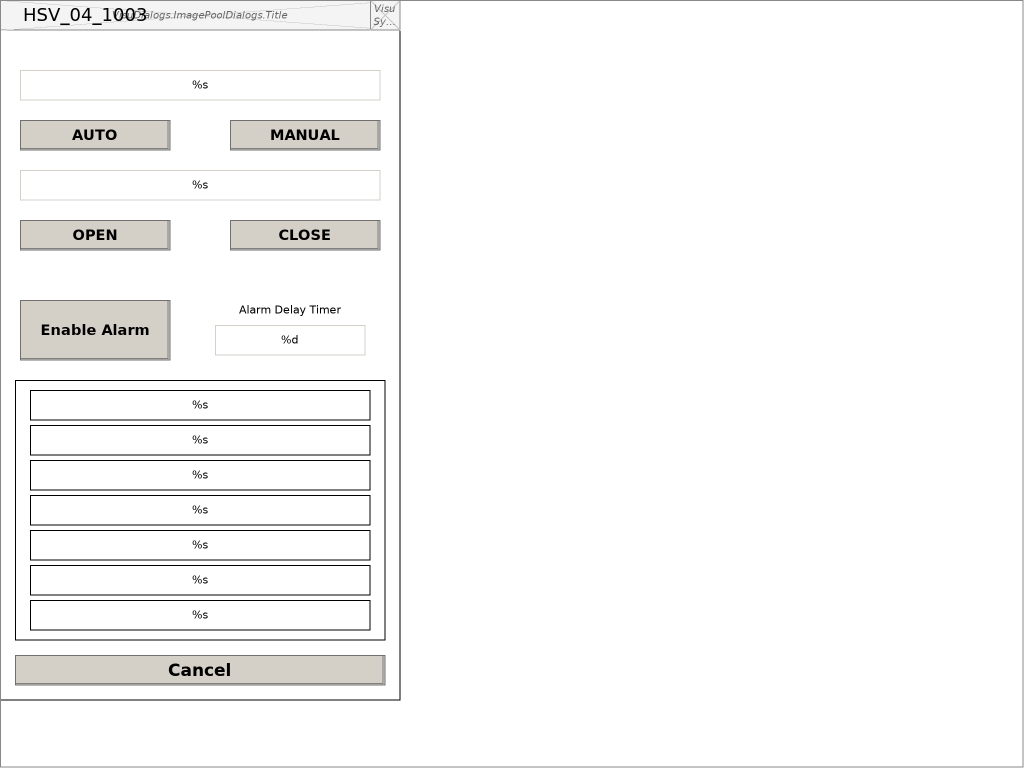
VISUALIZATION HSV_04_1003  // 1024x768
    Rectangle (0,0 400x700)
    Button (20,120 150x30), "AUTO"
        tap progHSVCntrl.HSV_04_1003.AutoReq
    Button (230,120 150x30), "MANUAL"
        tap progHSVCntrl.HSV_04_1003.ManReq
    Button (20,220 150x30), "OPEN"
        tap progHSVCntrl.HSV_04_1003.ManOpenReq
    Button (230,220 150x30), "CLOSE"
        tap progHSVCntrl.HSV_04_1003.ManCloseReq
    Textfield (20,70 360x30), "%s", text variable: progHSVCntrl.HSV_04_1003.strAutoMan
    Textfield (20,170 360x30), "%s", text variable: progHSVCntrl.HSV_04_1003.strOpenTravClose
    Button (20,300 150x60), "Enable Alarm"
        toggle progHSVCntrl.HSV_04_1003.EnableAlarm
    Textfield (215,325 150x30), "%d", text variable: progHSVCntrl.HSV_04_1003.AlarmDelayTime
    Label (215,295 150x30), "Alarm Delay Timer"
    Image (0,0 400x30), image: VisuDialogs.ImagePoolDialogs.Title
    Group (370,0 30x30)
        OnMouseClick: CloseDialog Dialog=HSV_04_1003, Result=OK, NumpadKeypadSet=True
        RoundedRectangle (0,0 30x30)
        Image (0,0 30x30), image: VisuSymbols.Symbols.Wrong
    Rectangle (15,380 370x260)
    RoundedRectangle (30,390 340x30), "%s", text variable: progHSVCntrl.HSV_04_1003.strInterlock_1
    RoundedRectangle (30,425 340x30), "%s", text variable: progHSVCntrl.HSV_04_1003.strInterlock_2
    RoundedRectangle (30,460 340x30), "%s", text variable: progHSVCntrl.HSV_04_1003.strInterlock_3
    RoundedRectangle (30,495 340x30), "%s", text variable: progHSVCntrl.HSV_04_1003.strInterlock_4
    RoundedRectangle (30,530 340x30), "%s", text variable: progHSVCntrl.HSV_04_1003.strInterlock_5
    RoundedRectangle (30,565 340x30), "%s", text variable: progHSVCntrl.HSV_04_1003.strInterlock_6
    RoundedRectangle (30,600 340x30), "%s", text variable: progHSVCntrl.HSV_04_1003.strInterlock_7
    Button (15,655 370x30), "Cancel"
        OnMouseClick: CloseDialog Dialog=HSV_04_1003, Result=OK, NumpadKeypadSet=True
    Label (20,0 210x30), "HSV_04_1003"
END_VISUALIZATION

// ---- VISUs/Diag/HSV/HSV_04_1004.TcVIS
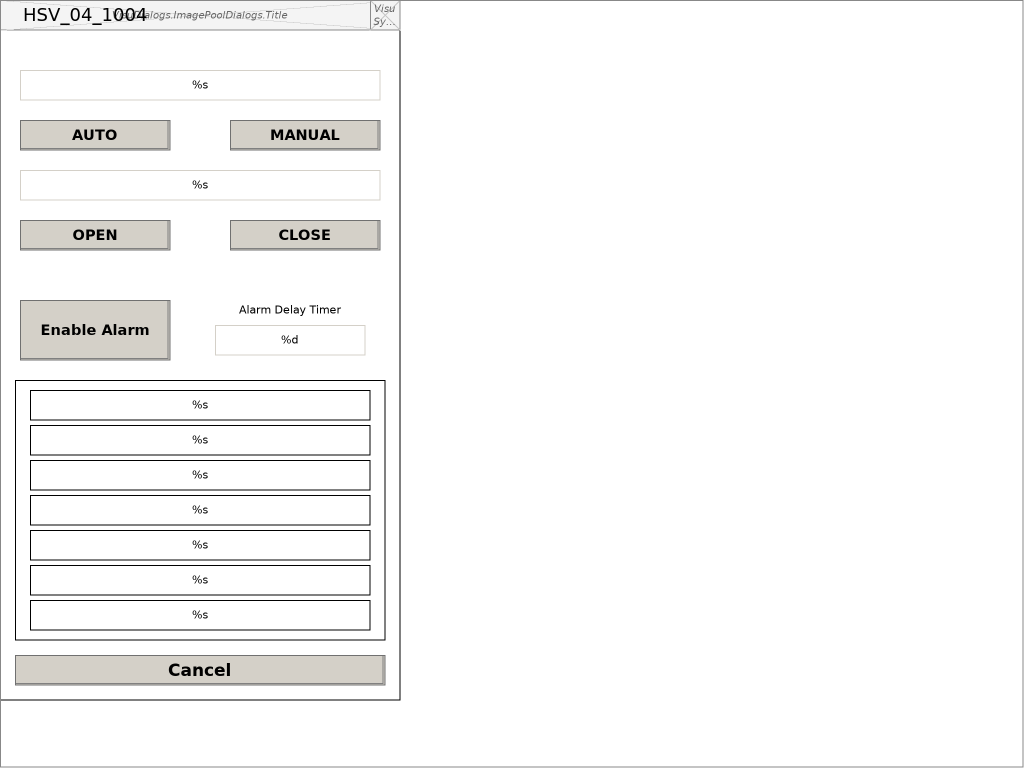
VISUALIZATION HSV_04_1004  // 1024x768
    Rectangle (0,0 400x700)
    Button (20,120 150x30), "AUTO"
        tap progHSVCntrl.HSV_04_1004.AutoReq
    Button (230,120 150x30), "MANUAL"
        tap progHSVCntrl.HSV_04_1004.ManReq
    Button (20,220 150x30), "OPEN"
        tap progHSVCntrl.HSV_04_1004.ManOpenReq
    Button (230,220 150x30), "CLOSE"
        tap progHSVCntrl.HSV_04_1004.ManCloseReq
    Textfield (20,70 360x30), "%s", text variable: progHSVCntrl.HSV_04_1004.strAutoMan
    Textfield (20,170 360x30), "%s", text variable: progHSVCntrl.HSV_04_1004.strOpenTravClose
    Button (20,300 150x60), "Enable Alarm"
        toggle progHSVCntrl.HSV_04_1004.EnableAlarm
    Textfield (215,325 150x30), "%d", text variable: progHSVCntrl.HSV_04_1004.AlarmDelayTime
    Label (215,295 150x30), "Alarm Delay Timer"
    Image (0,0 400x30), image: VisuDialogs.ImagePoolDialogs.Title
    Group (370,0 30x30)
        OnMouseClick: CloseDialog Dialog=HSV_04_1004, Result=OK, NumpadKeypadSet=True
        RoundedRectangle (0,0 30x30)
        Image (0,0 30x30), image: VisuSymbols.Symbols.Wrong
    Rectangle (15,380 370x260)
    RoundedRectangle (30,390 340x30), "%s", text variable: progHSVCntrl.HSV_04_1004.strInterlock_1
    RoundedRectangle (30,425 340x30), "%s", text variable: progHSVCntrl.HSV_04_1004.strInterlock_2
    RoundedRectangle (30,460 340x30), "%s", text variable: progHSVCntrl.HSV_04_1004.strInterlock_3
    RoundedRectangle (30,495 340x30), "%s", text variable: progHSVCntrl.HSV_04_1004.strInterlock_4
    RoundedRectangle (30,530 340x30), "%s", text variable: progHSVCntrl.HSV_04_1004.strInterlock_5
    RoundedRectangle (30,565 340x30), "%s", text variable: progHSVCntrl.HSV_04_1004.strInterlock_6
    RoundedRectangle (30,600 340x30), "%s", text variable: progHSVCntrl.HSV_04_1004.strInterlock_7
    Button (15,655 370x30), "Cancel"
        OnMouseClick: CloseDialog Dialog=HSV_04_1004, Result=OK, NumpadKeypadSet=True
    Label (20,0 210x30), "HSV_04_1004"
END_VISUALIZATION

// ---- VISUs/Diag/HSV/HSV_04_1005.TcVIS
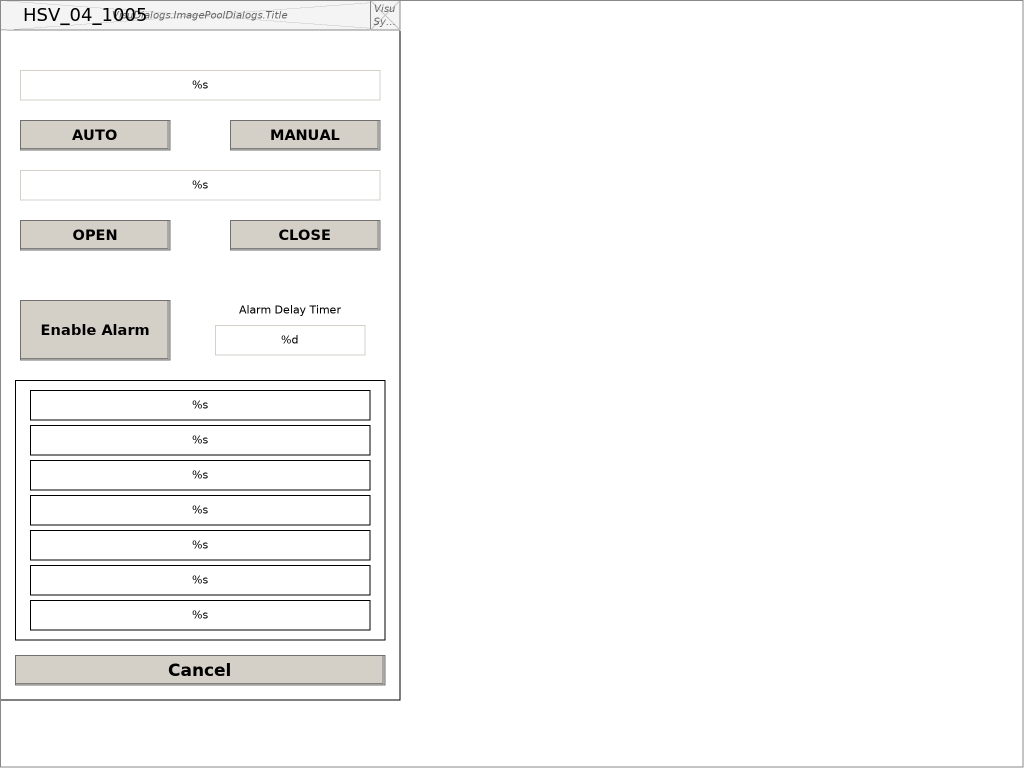
VISUALIZATION HSV_04_1005  // 1024x768
    Rectangle (0,0 400x700)
    Button (20,120 150x30), "AUTO"
        tap progHSVCntrl.HSV_04_1005.AutoReq
    Button (230,120 150x30), "MANUAL"
        tap progHSVCntrl.HSV_04_1005.ManReq
    Button (20,220 150x30), "OPEN"
        tap progHSVCntrl.HSV_04_1005.ManOpenReq
    Button (230,220 150x30), "CLOSE"
        tap progHSVCntrl.HSV_04_1005.ManCloseReq
    Textfield (20,70 360x30), "%s", text variable: progHSVCntrl.HSV_04_1005.strAutoMan
    Textfield (20,170 360x30), "%s", text variable: progHSVCntrl.HSV_04_1005.strOpenTravClose
    Button (20,300 150x60), "Enable Alarm"
        toggle progHSVCntrl.HSV_04_1005.EnableAlarm
    Textfield (215,325 150x30), "%d", text variable: progHSVCntrl.HSV_04_1005.AlarmDelayTime
    Label (215,295 150x30), "Alarm Delay Timer"
    Image (0,0 400x30), image: VisuDialogs.ImagePoolDialogs.Title
    Group (370,0 30x30)
        OnMouseClick: CloseDialog Dialog=HSV_04_1005, Result=OK, NumpadKeypadSet=True
        RoundedRectangle (0,0 30x30)
        Image (0,0 30x30), image: VisuSymbols.Symbols.Wrong
    Rectangle (15,380 370x260)
    RoundedRectangle (30,390 340x30), "%s", text variable: progHSVCntrl.HSV_04_1005.strInterlock_1
    RoundedRectangle (30,425 340x30), "%s", text variable: progHSVCntrl.HSV_04_1005.strInterlock_2
    RoundedRectangle (30,460 340x30), "%s", text variable: progHSVCntrl.HSV_04_1005.strInterlock_3
    RoundedRectangle (30,495 340x30), "%s", text variable: progHSVCntrl.HSV_04_1005.strInterlock_4
    RoundedRectangle (30,530 340x30), "%s", text variable: progHSVCntrl.HSV_04_1005.strInterlock_5
    RoundedRectangle (30,565 340x30), "%s", text variable: progHSVCntrl.HSV_04_1005.strInterlock_6
    RoundedRectangle (30,600 340x30), "%s", text variable: progHSVCntrl.HSV_04_1005.strInterlock_7
    Button (15,655 370x30), "Cancel"
        OnMouseClick: CloseDialog Dialog=HSV_04_1005, Result=OK, NumpadKeypadSet=True
    Label (20,0 210x30), "HSV_04_1005"
END_VISUALIZATION

// ---- VISUs/Diag/SCA/SCA_04_0100.TcVIS
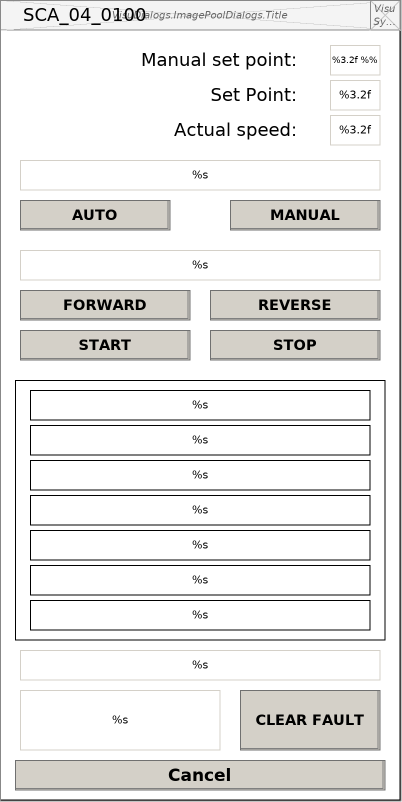
VISUALIZATION SCA_04_0100  // 402x802
    Rectangle (0,0 400x800)
    Button (20,200 150x30), "AUTO"
        tap progSCACntrl.SCA_04_0100.AutoReq
    Button (230,200 150x30), "MANUAL"
        tap progSCACntrl.SCA_04_0100.ManReq
    Button (20,290 170x30), "FORWARD"
        OnMouseClick: execute { progSCACntrl.SCA_04_0100.ManDirection := 0; }
    Button (210,290 170x30), "REVERSE"
        OnMouseClick: execute { progSCACntrl.SCA_04_0100.ManDirection := 1; }
    Textfield (20,160 360x30), "%s", text variable: progSCACntrl.SCA_04_0100.strAutoMan
    Textfield (20,250 360x30), "%s", text variable: progSCACntrl.SCA_04_0100.strStopTravRun
    Image (0,0 400x30), image: VisuDialogs.ImagePoolDialogs.Title
    Group (370,0 30x30)
        RoundedRectangle (0,0 30x30)
        Image (0,0 30x30), image: VisuSymbols.Symbols.Wrong
    Rectangle (15,380 370x260)
    RoundedRectangle (30,390 340x30), "%s", text variable: progSCACntrl.SCA_04_0100.strInterlock_1
    RoundedRectangle (30,425 340x30), "%s", text variable: progSCACntrl.SCA_04_0100.strInterlock_2
    RoundedRectangle (30,460 340x30), "%s", text variable: progSCACntrl.SCA_04_0100.strInterlock_3
    RoundedRectangle (30,495 340x30), "%s", text variable: progSCACntrl.SCA_04_0100.strInterlock_4
    RoundedRectangle (30,530 340x30), "%s", text variable: progSCACntrl.SCA_04_0100.strInterlock_5
    RoundedRectangle (30,565 340x30), "%s", text variable: progSCACntrl.SCA_04_0100.strInterlock_6
    RoundedRectangle (30,600 340x30), "%s", text variable: progSCACntrl.SCA_04_0100.strInterlock_7
    Button (15,760 370x30), "Cancel"
    Label (0,80 300x30), "Set Point:"
    Textfield (330,80 50x30), "%3.2f", text variable: progSCACntrl.SCA_04_0100.CommandSpeed
    Label (0,45 300x30), "Manual set point:"
    Textfield (330,45 50x30), "%3.2f %%", text variable: progSCACntrl.SCA_04_0100.ManSpeed
        OnMouseClick: write the text variable via VisuDialogs.Numpad, min progSCACntrl.SCA_04_0100.EngMin, max progSCACntrl.SCA_04_0100.EngMax, format %3.2f
    Label (0,115 300x30), "Actual speed:"
    Textfield (330,115 50x30), "%3.2f", text variable: progSCACntrl.SCA_04_0100.ActualSpeed
    Label (20,0 210x30), "SCA_04_0100"
    Button (20,330 170x30), "START"
        tap progSCACntrl.SCA_04_0100.ManStart
    Button (210,330 170x30), "STOP"
        tap progSCACntrl.SCA_04_0100.ManStop
    Textfield (20,650 360x30), "%s", text variable: progSCACntrl.SCA_04_0100.strAlmDesc
    Textfield (20,690 200x60), "%s", text variable: progSCACntrl.SCA_04_0100.strOKFault
    Button (240,690 140x60), "CLEAR FAULT"
        tap progSCACntrl.SCA_04_0100.ClearFlt
END_VISUALIZATION

// ---- VISUs/Screens/Overview.TcVIS
VISUALIZATION Overview  // 2x2
END_VISUALIZATION

// ---- VISUs/Screens/Vacuum_C1.TcVIS
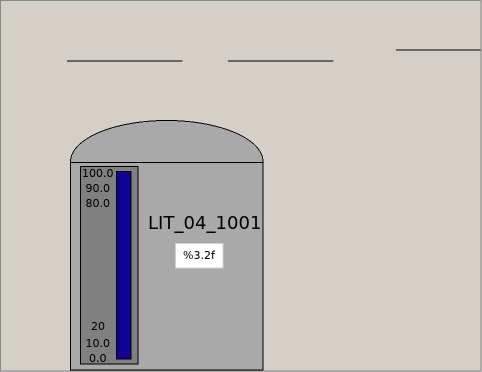
VISUALIZATION Vacuum_C1  // 482x372
    Line (182,61) (67,61)
    Line (333,61) (228,61)
    Line (480,50) (396,50)
    Group (70,120 200x250)
        Ellipse (0,0 193x83)
        Rectangle (0,42 193x208)
        Rectangle (10,46 58x198)
        Rectangle (46,51 15x188)
        Label (10,231 36x15), "0.0"
        Label (10,46 36x15), "100.0"
        Label (10,61 36x15), "90.0"
        Label (10,76 36x15), "80.0"
        Label (10,216 36x15), "10.0"
        Label (10,199 36x15), "20"
        Label (70,88 130x30), "LIT_04_1001"
        Textfield (105,123 48x25), "%3.2f", text variable: progLITCntrl.LIT_04_1001.Level
            OnMouseClick: write progLITCntrl.LIT_04_1001.Level via VisuDialogs.NumpadExtended, min 0.0, max 100.0
END_VISUALIZATION

// ---- VISUs/Templates/Diag/visuFCVDiag.TcVIS
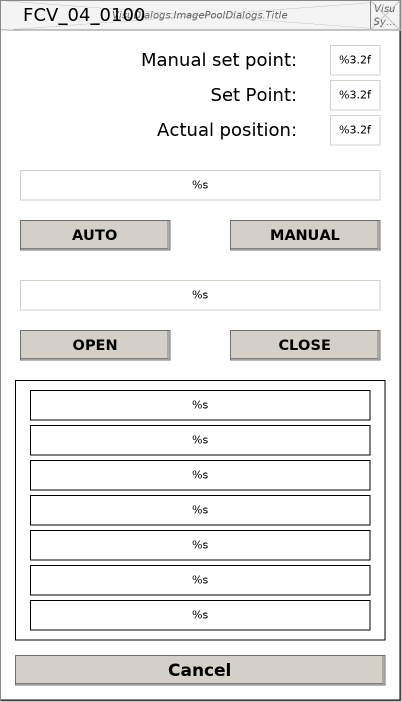
VISUALIZATION visuFCVDiag  // 402x702
    Rectangle (0,0 400x700)
    Button (20,220 150x30), "AUTO"
        tap progFCVCntrl.FCV_04_0100.AutoReq
    Button (230,220 150x30), "MANUAL"
        tap progFCVCntrl.FCV_04_0100.ManReq
    Button (20,330 150x30), "OPEN"
        tap progFCVCntrl.FCV_04_0100.ManOpenReq
    Button (230,330 150x30), "CLOSE"
        tap progFCVCntrl.FCV_04_0100.ManCloseReq
    Textfield (20,170 360x30), "%s", text variable: progFCVCntrl.FCV_04_0100.strAutoMan
    Textfield (20,280 360x30), "%s", text variable: progFCVCntrl.FCV_04_0100.strOpenTravClose
    Image (0,0 400x30), image: VisuDialogs.ImagePoolDialogs.Title
    Group (370,0 30x30)
        RoundedRectangle (0,0 30x30)
        Image (0,0 30x30), image: VisuSymbols.Symbols.Wrong
    Rectangle (15,380 370x260)
    RoundedRectangle (30,390 340x30), "%s", text variable: progFCVCntrl.FCV_04_0100.strInterlock_1
    RoundedRectangle (30,425 340x30), "%s", text variable: progFCVCntrl.FCV_04_0100.strInterlock_2
    RoundedRectangle (30,460 340x30), "%s", text variable: progFCVCntrl.FCV_04_0100.strInterlock_3
    RoundedRectangle (30,495 340x30), "%s", text variable: progFCVCntrl.FCV_04_0100.strInterlock_4
    RoundedRectangle (30,530 340x30), "%s", text variable: progFCVCntrl.FCV_04_0100.strInterlock_5
    RoundedRectangle (30,565 340x30), "%s", text variable: progFCVCntrl.FCV_04_0100.strInterlock_6
    RoundedRectangle (30,600 340x30), "%s", text variable: progFCVCntrl.FCV_04_0100.strInterlock_7
    Button (15,655 370x30), "Cancel"
    Label (0,80 300x30), "Set Point:"
    Textfield (330,80 50x30), "%3.2f", text variable: progFCVCntrl.FCV_04_0100.CmdSpOut
    Label (0,45 300x30), "Manual set point:"
    Textfield (330,45 50x30), "%3.2f", text variable: progFCVCntrl.FCV_04_0100.ManSP
        OnMouseClick: write progFCVCntrl.FCV_04_0100.ManSP via VisuDialogs.NumpadExtended
    Label (0,115 300x30), "Actual position:"
    Textfield (330,115 50x30), "%3.2f", text variable: progFCVCntrl.FCV_04_0100.ActPos
    Label (20,0 210x30), "FCV_04_0100"
END_VISUALIZATION

// ---- VISUs/Templates/Diag/visuHSVDiag.TcVIS
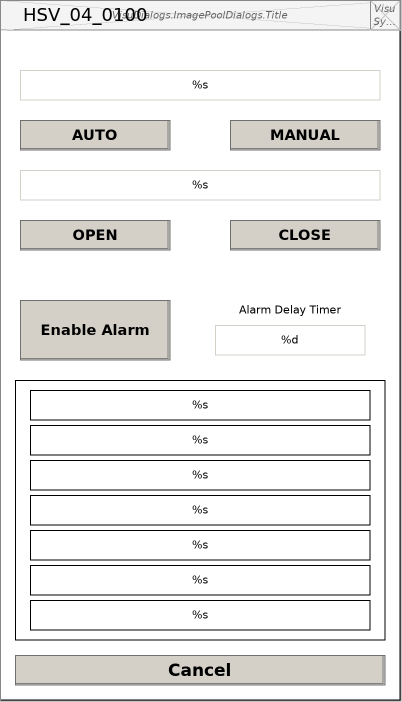
VISUALIZATION visuHSVDiag  // 402x702
    Rectangle (0,0 400x700)
    Button (20,120 150x30), "AUTO"
        tap progHSVCntrl.HSV_04_0100.AutoReq
    Button (230,120 150x30), "MANUAL"
        tap progHSVCntrl.HSV_04_0100.ManReq
    Button (20,220 150x30), "OPEN"
        tap progHSVCntrl.HSV_04_0100.ManOpenReq
    Button (230,220 150x30), "CLOSE"
        tap progHSVCntrl.HSV_04_0100.ManCloseReq
    Textfield (20,70 360x30), "%s", text variable: progHSVCntrl.HSV_04_0100.strAutoMan
    Textfield (20,170 360x30), "%s", text variable: progHSVCntrl.HSV_04_0100.strOpenTravClose
    Button (20,300 150x60), "Enable Alarm"
        toggle progHSVCntrl.HSV_04_0100.EnableAlarm
    Textfield (215,325 150x30), "%d"
    Label (215,295 150x30), "Alarm Delay Timer"
    Image (0,0 400x30), image: VisuDialogs.ImagePoolDialogs.Title
    Group (370,0 30x30)
        RoundedRectangle (0,0 30x30)
        Image (0,0 30x30), image: VisuSymbols.Symbols.Wrong
    Rectangle (15,380 370x260)
    RoundedRectangle (30,390 340x30), "%s", text variable: progHSVCntrl.HSV_04_0100.strInterlock_1
    RoundedRectangle (30,425 340x30), "%s", text variable: progHSVCntrl.HSV_04_0100.strInterlock_2
    RoundedRectangle (30,460 340x30), "%s", text variable: progHSVCntrl.HSV_04_0100.strInterlock_3
    RoundedRectangle (30,495 340x30), "%s", text variable: progHSVCntrl.HSV_04_0100.strInterlock_4
    RoundedRectangle (30,530 340x30), "%s", text variable: progHSVCntrl.HSV_04_0100.strInterlock_5
    RoundedRectangle (30,565 340x30), "%s", text variable: progHSVCntrl.HSV_04_0100.strInterlock_6
    RoundedRectangle (30,600 340x30), "%s", text variable: progHSVCntrl.HSV_04_0100.strInterlock_7
    Button (15,655 370x30), "Cancel"
    Label (20,0 210x30), "HSV_04_0100"
END_VISUALIZATION

// ---- VISUs/Templates/Diag/visuLITDiag.TcVIS
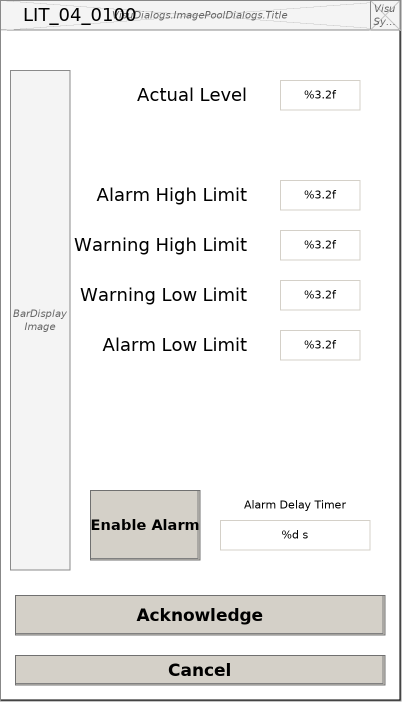
VISUALIZATION visuLITDiag  // 402x702
    Rectangle (0,0 400x700)
    Textfield (280,180 80x30), "%3.2f", text variable: progLITCntrl.LIT_04_0100.HHLimit
    Button (90,490 110x70), "Enable Alarm"
        toggle progHSVCntrl.HSV_04_0100.EnableAlarm
    Textfield (220,520 150x30), "%d s"
    Label (220,490 150x30), "Alarm Delay Timer"
    Image (0,0 400x30), image: VisuDialogs.ImagePoolDialogs.Title
    Group (370,0 30x30)
        RoundedRectangle (0,0 30x30)
        Image (0,0 30x30), image: VisuSymbols.Symbols.Wrong
    Button (15,655 370x30), "Cancel"
    Label (20,0 210x30), "LIT_04_0100"
    Label (0,180 250x30), "Alarm High Limit"
    Label (0,230 250x30), "Warning High Limit"
    Label (0,280 250x30), "Warning Low Limit"
    Label (0,330 250x30), "Alarm Low Limit"
    Textfield (280,230 80x30), "%3.2f", text variable: progLITCntrl.LIT_04_0100.HLimit
    Textfield (280,280 80x30), "%3.2f", text variable: progLITCntrl.LIT_04_0100.LLimit
    Textfield (280,330 80x30), "%3.2f", text variable: progLITCntrl.LIT_04_0100.LLLimit
    Button (15,595 370x40), "Acknowledge"
    Textfield (280,80 80x30), "%3.2f", text variable: progLITCntrl.LIT_04_0100.Level
    Label (0,80 250x30), "Actual Level"
    BarDisplayImage (10,70 60x500), value: progLITCntrl.LIT_04_0100.Level, style: BarDisplayImage-Gray, scale format: %.1f, scale 0..100
END_VISUALIZATION

// ---- VISUs/Templates/Diag/visuPITDiag.TcVIS
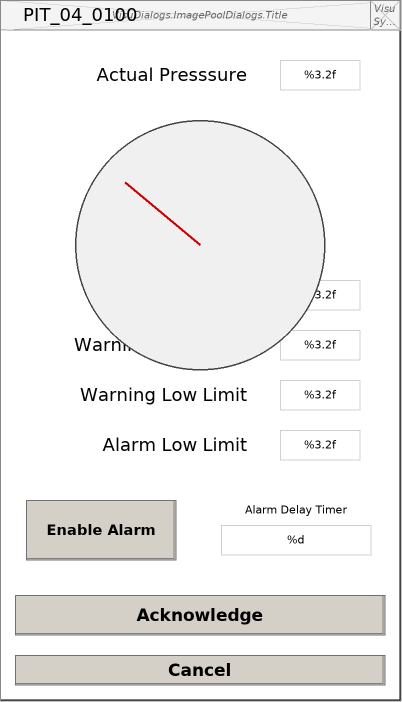
VISUALIZATION visuPITDiag  // 402x702
    Rectangle (0,0 400x700)
    Textfield (280,280 80x30), "%3.2f"
    Button (26,500 150x60), "Enable Alarm"
        toggle progHSVCntrl.HSV_04_0100.EnableAlarm
    Textfield (221,525 150x30), "%d"
    Label (221,495 150x30), "Alarm Delay Timer"
    Image (0,0 400x30), image: VisuDialogs.ImagePoolDialogs.Title
    Group (370,0 30x30)
        RoundedRectangle (0,0 30x30)
        Image (0,0 30x30), image: VisuSymbols.Symbols.Wrong
    Button (15,655 370x30), "Cancel"
    Label (20,0 210x30), "PIT_04_0100"
    Label (0,280 250x30), "Alarm High Limit"
    Label (0,330 250x30), "Warning High Limit"
    Label (0,380 250x30), "Warning Low Limit"
    Label (0,430 250x30), "Alarm Low Limit"
    Textfield (280,330 80x30), "%3.2f"
    Textfield (280,380 80x30), "%3.2f"
    Textfield (280,430 80x30), "%3.2f"
    Button (15,595 370x40), "Acknowledge"
    Textfield (280,60 80x30), "%3.2f"
    Label (0,60 250x30), "Actual Presssure"
    Meter180 (75,120 250x250), style: Meter-Meter180-Gray, scale format: %.1f, scale 0..100
END_VISUALIZATION

// ---- VISUs/Templates/Diag/visuSCADiag.TcVIS
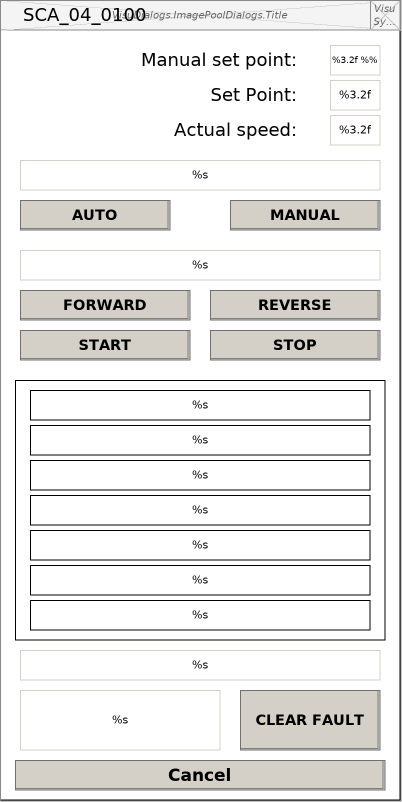
VISUALIZATION visuSCADiag  // 402x802
    Rectangle (0,0 400x800)
    Button (20,200 150x30), "AUTO"
        tap progSCACntrl.SCA_04_0100.AutoReq
    Button (230,200 150x30), "MANUAL"
        tap progSCACntrl.SCA_04_0100.ManReq
    Button (20,290 170x30), "FORWARD"
        OnMouseClick: execute { progSCACntrl.SCA_04_0100.ManDirection := 0; }
    Button (210,290 170x30), "REVERSE"
        OnMouseClick: execute { progSCACntrl.SCA_04_0100.ManDirection := 1; }
    Textfield (20,160 360x30), "%s", text variable: progSCACntrl.SCA_04_0100.strAutoMan
    Textfield (20,250 360x30), "%s", text variable: progSCACntrl.SCA_04_0100.strStopTravRun
    Image (0,0 400x30), image: VisuDialogs.ImagePoolDialogs.Title
    Group (370,0 30x30)
        RoundedRectangle (0,0 30x30)
        Image (0,0 30x30), image: VisuSymbols.Symbols.Wrong
    Rectangle (15,380 370x260)
    RoundedRectangle (30,390 340x30), "%s", text variable: progSCACntrl.SCA_04_0100.strInterlock_1
    RoundedRectangle (30,425 340x30), "%s", text variable: progSCACntrl.SCA_04_0100.strInterlock_2
    RoundedRectangle (30,460 340x30), "%s", text variable: progSCACntrl.SCA_04_0100.strInterlock_3
    RoundedRectangle (30,495 340x30), "%s", text variable: progSCACntrl.SCA_04_0100.strInterlock_4
    RoundedRectangle (30,530 340x30), "%s", text variable: progSCACntrl.SCA_04_0100.strInterlock_5
    RoundedRectangle (30,565 340x30), "%s", text variable: progSCACntrl.SCA_04_0100.strInterlock_6
    RoundedRectangle (30,600 340x30), "%s", text variable: progSCACntrl.SCA_04_0100.strInterlock_7
    Button (15,760 370x30), "Cancel"
    Label (0,80 300x30), "Set Point:"
    Textfield (330,80 50x30), "%3.2f", text variable: progSCACntrl.SCA_04_0100.CommandSpeed
    Label (0,45 300x30), "Manual set point:"
    Textfield (330,45 50x30), "%3.2f %%", text variable: progSCACntrl.SCA_04_0100.ManSpeed
        OnMouseClick: write the text variable via VisuDialogs.Numpad, min progSCACntrl.SCA_04_0100.EngMin, max progSCACntrl.SCA_04_0100.EngMax, format %3.2f
    Label (0,115 300x30), "Actual speed:"
    Textfield (330,115 50x30), "%3.2f", text variable: progSCACntrl.SCA_04_0100.ActualSpeed
    Label (20,0 210x30), "SCA_04_0100"
    Button (20,330 170x30), "START"
        tap progSCACntrl.SCA_04_0100.ManStart
    Button (210,330 170x30), "STOP"
        tap progSCACntrl.SCA_04_0100.ManStop
    Textfield (20,650 360x30), "%s", text variable: progSCACntrl.SCA_04_0100.strAlmDesc
    Textfield (20,690 200x60), "%s", text variable: progSCACntrl.SCA_04_0100.strOKFault
    Button (240,690 140x60), "CLEAR FAULT"
        tap progSCACntrl.SCA_04_0100.ClearFlt
END_VISUALIZATION

// ---- VISUs/Templates/Diag/visuTITDiag.TcVIS
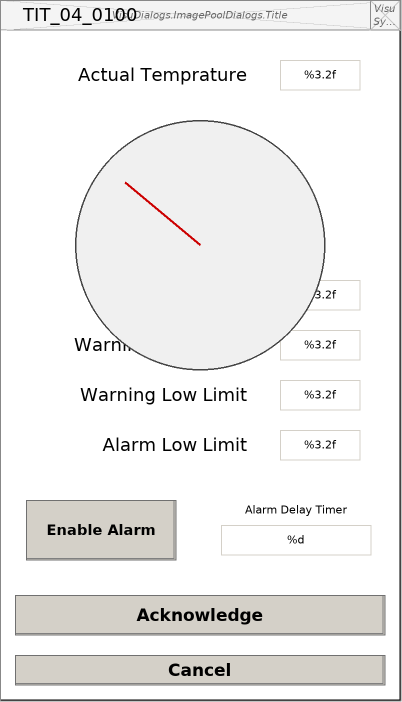
VISUALIZATION visuTITDiag  // 402x702
    Rectangle (0,0 400x700)
    Textfield (280,280 80x30), "%3.2f"
    Button (26,500 150x60), "Enable Alarm"
        toggle progHSVCntrl.HSV_04_0100.EnableAlarm
    Textfield (221,525 150x30), "%d"
    Label (221,495 150x30), "Alarm Delay Timer"
    Image (0,0 400x30), image: VisuDialogs.ImagePoolDialogs.Title
    Group (370,0 30x30)
        RoundedRectangle (0,0 30x30)
        Image (0,0 30x30), image: VisuSymbols.Symbols.Wrong
    Button (15,655 370x30), "Cancel"
    Label (20,0 210x30), "TIT_04_0100"
    Label (0,280 250x30), "Alarm High Limit"
    Label (0,330 250x30), "Warning High Limit"
    Label (0,380 250x30), "Warning Low Limit"
    Label (0,430 250x30), "Alarm Low Limit"
    Textfield (280,330 80x30), "%3.2f"
    Textfield (280,380 80x30), "%3.2f"
    Textfield (280,430 80x30), "%3.2f"
    Button (15,595 370x40), "Acknowledge"
    Textfield (280,60 80x30), "%3.2f"
    Label (0,60 250x30), "Actual Temprature"
    Meter180 (75,120 250x250), style: Meter-Meter180-Gray, scale format: %.1f, scale 0..100
END_VISUALIZATION

// ---- VISUs/Templates/inDevelopment/visuServoDiag.TcVIS
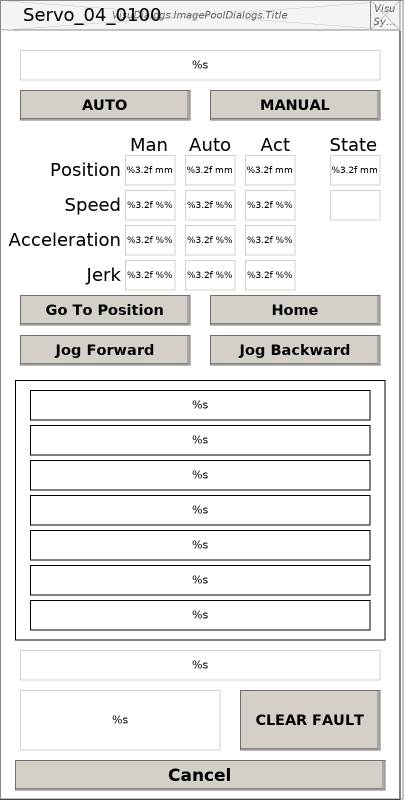
VISUALIZATION visuServoDiag  // 404x800
    Rectangle (0,0 400x800)
    Button (20,90 170x30), "AUTO"
        tap progServoCntrl.Servo_04_0100.AutoReq
    Button (210,90 170x30), "MANUAL"
        tap progServoCntrl.Servo_04_0100.ManReq
    Textfield (20,50 360x30), "%s", text variable: progServoCntrl.Servo_04_0100.strAutoMan
    Image (0,0 400x30), image: VisuDialogs.ImagePoolDialogs.Title
    Group (370,0 30x30)
        RoundedRectangle (0,0 30x30)
        Image (0,0 30x30), image: VisuSymbols.Symbols.Wrong
    Rectangle (15,380 370x260)
    RoundedRectangle (30,390 340x30), "%s", text variable: progSCACntrl.SCA_04_0100.strInterlock_1
    RoundedRectangle (30,425 340x30), "%s", text variable: progSCACntrl.SCA_04_0100.strInterlock_2
    RoundedRectangle (30,460 340x30), "%s", text variable: progSCACntrl.SCA_04_0100.strInterlock_3
    RoundedRectangle (30,495 340x30), "%s", text variable: progSCACntrl.SCA_04_0100.strInterlock_4
    RoundedRectangle (30,530 340x30), "%s", text variable: progSCACntrl.SCA_04_0100.strInterlock_5
    RoundedRectangle (30,565 340x30), "%s", text variable: progSCACntrl.SCA_04_0100.strInterlock_6
    RoundedRectangle (30,600 340x30), "%s", text variable: progSCACntrl.SCA_04_0100.strInterlock_7
    Button (15,760 370x30), "Cancel"
    Label (115,130 56x30), "Man"
    Textfield (125,155 50x30), "%3.2f mm", text variable: progServoCntrl.Servo_04_0100.ManPosSP
        OnMouseClick: write the text variable via VisuDialogs.Numpad, min progSCACntrl.SCA_04_0100.EngMin, max progSCACntrl.SCA_04_0100.EngMax, format %3.2f
    Label (20,0 210x30), "Servo_04_0100"
    Button (20,295 170x30), "Go To Position"
        tap progServoCntrl.Servo_04_0100.GoToPosition
    Textfield (20,650 360x30), "%s", text variable: progServoCntrl.Servo_04_0100.Faulted
    Textfield (20,690 200x60), "%s", text variable: progServoCntrl.Servo_04_0100.FaultID
    Button (240,690 140x60), "CLEAR FAULT"
        tap progServoCntrl.Servo_04_0100.ClearFault
    Label (180,130 54x30), "Auto"
    Label (255,130 38x30), "Act"
    Textfield (125,190 50x30), "%3.2f %%", text variable: progServoCntrl.Servo_04_0100.ManSpeedSP
        OnMouseClick: write the text variable via VisuDialogs.Numpad, min progSCACntrl.SCA_04_0100.EngMin, max progSCACntrl.SCA_04_0100.EngMax, format %3.2f
    Label (45,155 79x30), "Position"
    Label (45,190 79x30), "Speed"
    Label (-4,225 128x30), "Acceleration"
    Label (45,260 79x30), "Jerk"
    Textfield (125,225 50x30), "%3.2f %%", text variable: progServoCntrl.Servo_04_0100.ManAccSP
        OnMouseClick: write the text variable via VisuDialogs.Numpad, min progSCACntrl.SCA_04_0100.EngMin, max progSCACntrl.SCA_04_0100.EngMax, format %3.2f
    Textfield (125,260 50x30), "%3.2f %%", text variable: progServoCntrl.Servo_04_0100.ManJerk
        OnMouseClick: write the text variable via VisuDialogs.Numpad, min progSCACntrl.SCA_04_0100.EngMin, max progSCACntrl.SCA_04_0100.EngMax, format %3.2f
    Textfield (185,155 50x30), "%3.2f mm", text variable: progServoCntrl.Servo_04_0100.AutoPosSp
        OnMouseClick: write the text variable via VisuDialogs.Numpad, min progSCACntrl.SCA_04_0100.EngMin, max progSCACntrl.SCA_04_0100.EngMax, format %3.2f
    Textfield (185,190 50x30), "%3.2f %%", text variable: progServoCntrl.Servo_04_0100.AutoSpeedSp
        OnMouseClick: write the text variable via VisuDialogs.Numpad, min progSCACntrl.SCA_04_0100.EngMin, max progSCACntrl.SCA_04_0100.EngMax, format %3.2f
    Textfield (185,225 50x30), "%3.2f %%", text variable: progServoCntrl.Servo_04_0100.AutoAccSp
        OnMouseClick: write the text variable via VisuDialogs.Numpad, min progSCACntrl.SCA_04_0100.EngMin, max progSCACntrl.SCA_04_0100.EngMax, format %3.2f
    Textfield (185,260 50x30), "%3.2f %%", text variable: progServoCntrl.Servo_04_0100.AutoJerkSp
        OnMouseClick: write the text variable via VisuDialogs.Numpad, min progSCACntrl.SCA_04_0100.EngMin, max progSCACntrl.SCA_04_0100.EngMax, format %3.2f
    Textfield (245,155 50x30), "%3.2f mm", text variable: progServoCntrl.Servo_04_0100.PosSP
        OnMouseClick: write the text variable via VisuDialogs.Numpad, min progSCACntrl.SCA_04_0100.EngMin, max progSCACntrl.SCA_04_0100.EngMax, format %3.2f
    Textfield (245,190 50x30), "%3.2f %%", text variable: progServoCntrl.Servo_04_0100.SpeedSP
        OnMouseClick: write the text variable via VisuDialogs.Numpad, min progSCACntrl.SCA_04_0100.EngMin, max progSCACntrl.SCA_04_0100.EngMax, format %3.2f
    Textfield (245,225 50x30), "%3.2f %%", text variable: progServoCntrl.Servo_04_0100.AccSP
        OnMouseClick: write the text variable via VisuDialogs.Numpad, min progSCACntrl.SCA_04_0100.EngMin, max progSCACntrl.SCA_04_0100.EngMax, format %3.2f
    Textfield (245,260 50x30), "%3.2f %%", text variable: progServoCntrl.Servo_04_0100.JerkSP
        OnMouseClick: write the text variable via VisuDialogs.Numpad, min progSCACntrl.SCA_04_0100.EngMin, max progSCACntrl.SCA_04_0100.EngMax, format %3.2f
    Button (210,295 170x30), "Home"
        tap progServoCntrl.Servo_04_0100.HomeReq
    Button (20,335 170x30), "Jog Forward"
        tap progServoCntrl.Servo_04_0100.JogForward
    Button (210,335 170x30), "Jog Backward"
        tap progServoCntrl.Servo_04_0100.JogBackward
    Label (320,130 60x30), "State"
    Textfield (330,155 50x30), "%3.2f mm", text variable: progServoCntrl.Servo_04_0100.Position
        OnMouseClick: write the text variable via VisuDialogs.Numpad, min progSCACntrl.SCA_04_0100.EngMin, max progSCACntrl.SCA_04_0100.EngMax, format %3.2f
    Textfield (330,190 50x30), text variable: progServoCntrl.Servo_04_0100.Speed
        OnMouseClick: write the text variable via VisuDialogs.Numpad, min progSCACntrl.SCA_04_0100.EngMin, max progSCACntrl.SCA_04_0100.EngMax, format %3.2f
END_VISUALIZATION

// ---- VISUs/Templates/Sym/Vessel.TcVIS
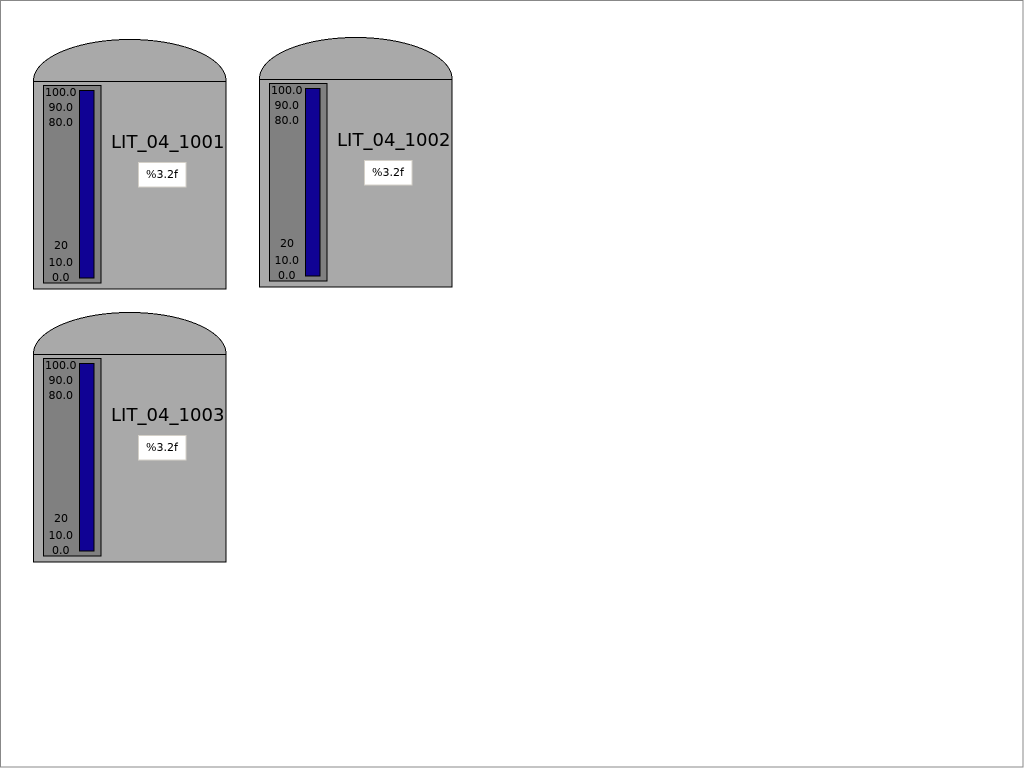
VISUALIZATION Vessel  // 1024x768
    Group (33,39 200x250)
        Ellipse (0,0 193x83)
        Rectangle (0,42 193x208)
        Rectangle (10,46 58x198)
        Rectangle (46,51 15x188)
        Label (10,231 36x15), "0.0"
        Label (10,46 36x15), "100.0"
        Label (10,61 36x15), "90.0"
        Label (10,76 36x15), "80.0"
        Label (10,216 36x15), "10.0"
        Label (10,199 36x15), "20"
        Label (70,88 130x30), "LIT_04_1001"
        Textfield (105,123 48x25), "%3.2f", text variable: progLITCntrl.LIT_04_1001.Level
            OnMouseClick: write progLITCntrl.LIT_04_1001.Level via VisuDialogs.NumpadExtended, min 0.0, max 100.0
    Group (259,37 200x250)
        Ellipse (0,0 193x83)
        Rectangle (0,42 193x208)
        Rectangle (10,46 58x198)
        Rectangle (46,51 15x188)
        Label (10,231 36x15), "0.0"
        Label (10,46 36x15), "100.0"
        Label (10,61 36x15), "90.0"
        Label (10,76 36x15), "80.0"
        Label (10,216 36x15), "10.0"
        Label (10,199 36x15), "20"
        Label (70,88 130x30), "LIT_04_1002"
        Textfield (105,123 48x25), "%3.2f", text variable: progLITCntrl.LIT_04_1002.Level
            OnMouseClick: write progLITCntrl.LIT_04_1002.Level via VisuDialogs.NumpadExtended, min 0.0, max 100.0
    Group (33,312 200x250)
        Ellipse (0,0 193x83)
        Rectangle (0,42 193x208)
        Rectangle (10,46 58x198)
        Rectangle (46,51 15x188)
        Label (10,231 36x15), "0.0"
        Label (10,46 36x15), "100.0"
        Label (10,61 36x15), "90.0"
        Label (10,76 36x15), "80.0"
        Label (10,216 36x15), "10.0"
        Label (10,199 36x15), "20"
        Label (70,88 130x30), "LIT_04_1003"
        Textfield (105,123 48x25), "%3.2f", text variable: progLITCntrl.LIT_04_1003.Level
            OnMouseClick: write progLITCntrl.LIT_04_1003.Level via VisuDialogs.NumpadExtended, min 0.0, max 100.0
END_VISUALIZATION

// ---- VISUs/Templates/Sym/visuHSVSim.TcVIS
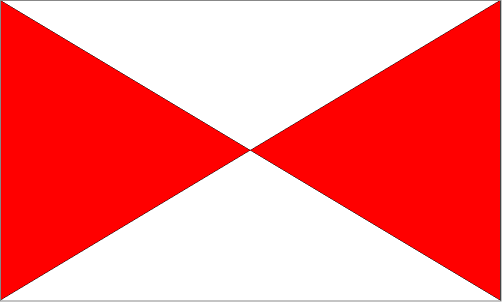
VISUALIZATION visuHSVSim  // 502x302
    Group (0,0 500x300)
        Polygon (0,0) (0,300) (250,150), invisible if: NOT progHSVCntrl.HSV_04_0100.FB_Close
        Polygon (500,0) (500,300) (250,150), invisible if: NOT progHSVCntrl.HSV_04_0100.FB_Close
        Polygon (0,0) (0,300) (250,150), invisible if: NOT progHSVCntrl.HSV_04_0100.FB_Travelling
        Polygon (500,0) (500,300) (250,150), invisible if: NOT progHSVCntrl.HSV_04_0100.FB_Travelling
        Polygon (0,0) (0,300) (250,150), invisible if: NOT progHSVCntrl.HSV_04_0100.FB_Open
        Polygon (500,0) (500,300) (250,150), invisible if: NOT progHSVCntrl.HSV_04_0100.FB_Open
        Polygon (0,0) (0,300) (250,150), invisible if: NOT progHSVCntrl.HSV_04_0100.Alarm
        Polygon (500,0) (500,300) (250,150), invisible if: NOT progHSVCntrl.HSV_04_0100.Alarm
END_VISUALIZATION

// ---- VISUs/Templates/Sym/visuFCVSim.TcVIS
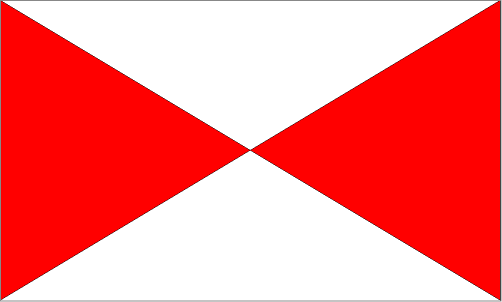
VISUALIZATION visuFCVSim  // 502x302
    Polygon (0,0) (0,300) (250,150), invisible if: NOT progFCVCntrl.FCV_04_0100.FB_Close
    Polygon (500,0) (500,300) (250,150), invisible if: NOT progFCVCntrl.FCV_04_0100.FB_Close
    Polygon (0,0) (0,300) (250,150), invisible if: NOT progFCVCntrl.FCV_04_0100.FB_Travelling
    Polygon (500,0) (500,300) (250,150), invisible if: NOT progFCVCntrl.FCV_04_0100.FB_Travelling
    Polygon (0,0) (0,300) (250,150), invisible if: NOT progFCVCntrl.FCV_04_0100.FB_Open
    Polygon (500,0) (500,300) (250,150), invisible if: NOT progFCVCntrl.FCV_04_0100.FB_Open
    Polygon (0,0) (0,300) (250,150), invisible if: NOT progFCVCntrl.FCV_04_0100.Alarm
    Polygon (500,0) (500,300) (250,150), invisible if: NOT progFCVCntrl.FCV_04_0100.Alarm
END_VISUALIZATION

// ---- VISUs/TrialAndError/visu.TcVIS
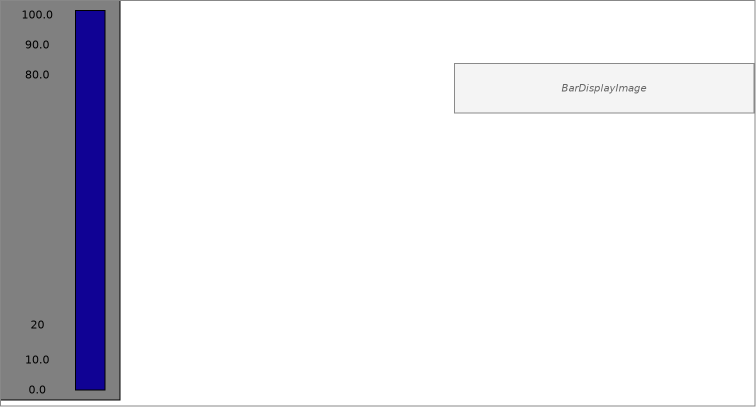
VISUALIZATION visu  // 756x407
    BarDisplayImage (454,63 300x50), style: BarDisplayImage-Gray, scale format: %.1f, scale 0..100
    Rectangle (0,0 120x400)
    Rectangle (75,10 30x380)
    Label (0,375 75x30), "0.0"
    Label (0,0 75x30), "100.0"
    Label (0,30 75x30), "90.0"
    Label (0,60 75x30), "80.0"
    Label (0,345 75x30), "10.0"
    Label (0,310 75x30), "20"
END_VISUALIZATION

// ---- VISUs/TrialAndError/Visualization.TcVIS
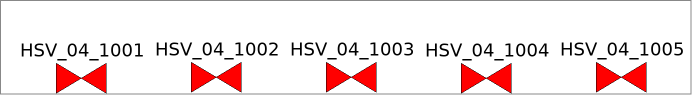
VISUALIZATION Visualization  // 692x95
    Group (15,24 135x69)
        OnMouseClick: OpenDialog Dialog=HSV_04_1001, OpenModal=True, OpenCentered=True
        Polygon (41,39) (41,69) (66,54), invisible if: NOT progHSVCntrl.HSV_04_1001.FB_Close
        Polygon (91,39) (91,69) (66,54), invisible if: NOT progHSVCntrl.HSV_04_1001.FB_Close
        Polygon (41,39) (41,69) (66,54), invisible if: NOT progHSVCntrl.HSV_04_1001.FB_Travelling
        Polygon (91,39) (91,69) (66,54), invisible if: NOT progHSVCntrl.HSV_04_1001.FB_Travelling
        Polygon (41,39) (41,69) (66,54), invisible if: NOT progHSVCntrl.HSV_04_1001.FB_Open
        Polygon (91,39) (91,69) (66,54), invisible if: NOT progHSVCntrl.HSV_04_1001.FB_Open
        Polygon (41,39) (41,69) (66,54), invisible if: NOT progHSVCntrl.HSV_04_1001.Alarm
        Polygon (91,39) (91,69) (66,54), invisible if: NOT progHSVCntrl.HSV_04_1001.Alarm
        Label (0,0 135x53), "HSV_04_1001"
    Group (150,23 135x69)
        OnMouseClick: OpenDialog Dialog=HSV_04_1002, OpenModal=True, OpenCentered=True
        Polygon (41,39) (41,69) (66,54), invisible if: NOT progHSVCntrl.HSV_04_1002.FB_Close
        Polygon (91,39) (91,69) (66,54), invisible if: NOT progHSVCntrl.HSV_04_1002.FB_Close
        Polygon (41,39) (41,69) (66,54), invisible if: NOT progHSVCntrl.HSV_04_1002.FB_Travelling
        Polygon (91,39) (91,69) (66,54), invisible if: NOT progHSVCntrl.HSV_04_1002.FB_Travelling
        Polygon (41,39) (41,69) (66,54), invisible if: NOT progHSVCntrl.HSV_04_1002.FB_Open
        Polygon (91,39) (91,69) (66,54), invisible if: NOT progHSVCntrl.HSV_04_1002.FB_Open
        Polygon (41,39) (41,69) (66,54), invisible if: NOT progHSVCntrl.HSV_04_1002.Alarm
        Polygon (91,39) (91,69) (66,54), invisible if: NOT progHSVCntrl.HSV_04_1002.Alarm
        Label (0,0 135x53), "HSV_04_1002"
    Group (285,23 135x69)
        OnMouseClick: OpenDialog Dialog=HSV_04_1003, OpenModal=True, OpenCentered=True
        Polygon (41,39) (41,69) (66,54), invisible if: NOT progHSVCntrl.HSV_04_1003.FB_Close
        Polygon (91,39) (91,69) (66,54), invisible if: NOT progHSVCntrl.HSV_04_1003.FB_Close
        Polygon (41,39) (41,69) (66,54), invisible if: NOT progHSVCntrl.HSV_04_1003.FB_Travelling
        Polygon (91,39) (91,69) (66,54), invisible if: NOT progHSVCntrl.HSV_04_1003.FB_Travelling
        Polygon (41,39) (41,69) (66,54), invisible if: NOT progHSVCntrl.HSV_04_1003.FB_Open
        Polygon (91,39) (91,69) (66,54), invisible if: NOT progHSVCntrl.HSV_04_1003.FB_Open
        Polygon (41,39) (41,69) (66,54), invisible if: NOT progHSVCntrl.HSV_04_1003.Alarm
        Polygon (91,39) (91,69) (66,54), invisible if: NOT progHSVCntrl.HSV_04_1003.Alarm
        Label (0,0 135x53), "HSV_04_1003"
    Group (420,24 135x69)
        OnMouseClick: OpenDialog Dialog=HSV_04_1004, OpenModal=True, OpenCentered=True
        Polygon (41,39) (41,69) (66,54), invisible if: NOT progHSVCntrl.HSV_04_1004.FB_Close
        Polygon (91,39) (91,69) (66,54), invisible if: NOT progHSVCntrl.HSV_04_1004.FB_Close
        Polygon (41,39) (41,69) (66,54), invisible if: NOT progHSVCntrl.HSV_04_1004.FB_Travelling
        Polygon (91,39) (91,69) (66,54), invisible if: NOT progHSVCntrl.HSV_04_1004.FB_Travelling
        Polygon (41,39) (41,69) (66,54), invisible if: NOT progHSVCntrl.HSV_04_1004.FB_Open
        Polygon (91,39) (91,69) (66,54), invisible if: NOT progHSVCntrl.HSV_04_1004.FB_Open
        Polygon (41,39) (41,69) (66,54), invisible if: NOT progHSVCntrl.HSV_04_1004.Alarm
        Polygon (91,39) (91,69) (66,54), invisible if: NOT progHSVCntrl.HSV_04_1004.Alarm
        Label (0,0 135x53), "HSV_04_1004"
    Group (555,23 135x69)
        Polygon (41,39) (41,69) (66,54), invisible if: NOT progHSVCntrl.HSV_04_1005.FB_Close
        Polygon (91,39) (91,69) (66,54), invisible if: NOT progHSVCntrl.HSV_04_1005.FB_Close
        Polygon (41,39) (41,69) (66,54), invisible if: NOT progHSVCntrl.HSV_04_1005.FB_Travelling
        Polygon (91,39) (91,69) (66,54), invisible if: NOT progHSVCntrl.HSV_04_1005.FB_Travelling
        Polygon (41,39) (41,69) (66,54), invisible if: NOT progHSVCntrl.HSV_04_1005.FB_Open
        Polygon (91,39) (91,69) (66,54), invisible if: NOT progHSVCntrl.HSV_04_1005.FB_Open
        Polygon (41,39) (41,69) (66,54), invisible if: NOT progHSVCntrl.HSV_04_1005.Alarm
        Polygon (91,39) (91,69) (66,54), invisible if: NOT progHSVCntrl.HSV_04_1005.Alarm
        Label (0,0 135x53), "HSV_04_1005"
END_VISUALIZATION
